{attribute 'qualified_only'}
{attribute 'strict'}
TYPE E_StatusSettings :
(
	enum_member := 0
);
END_TYPE

(* stored: Version 1.1.0.1, ProductVersion 3.1.4024.12
   DUT E_StatusSettings: Id {cbbc3ac6-3758-4a70-ae9b-379c1a508d22} *)
